PROGRAM main
VAR
	ButtonON_LED AT %IX100.0 : bool;
	ButtonOFF_LED AT %IX100.1 : bool;
	ButtonON_LEDBlink AT %IX100.2 : bool;
	ButtonOFF_LEDBlink AT %IX100.3 : bool;
	LED1 AT %QX100.0 : bool;
	LED2 AT %QX100.1 : bool;
	LED3 AT %QX100.2 : bool;
	Start_Blink : bool;
	TON0_Coil : bool;
	TON1_Coil : bool;
	TON0 : TON;
	TON1 : TON;
END_VAR

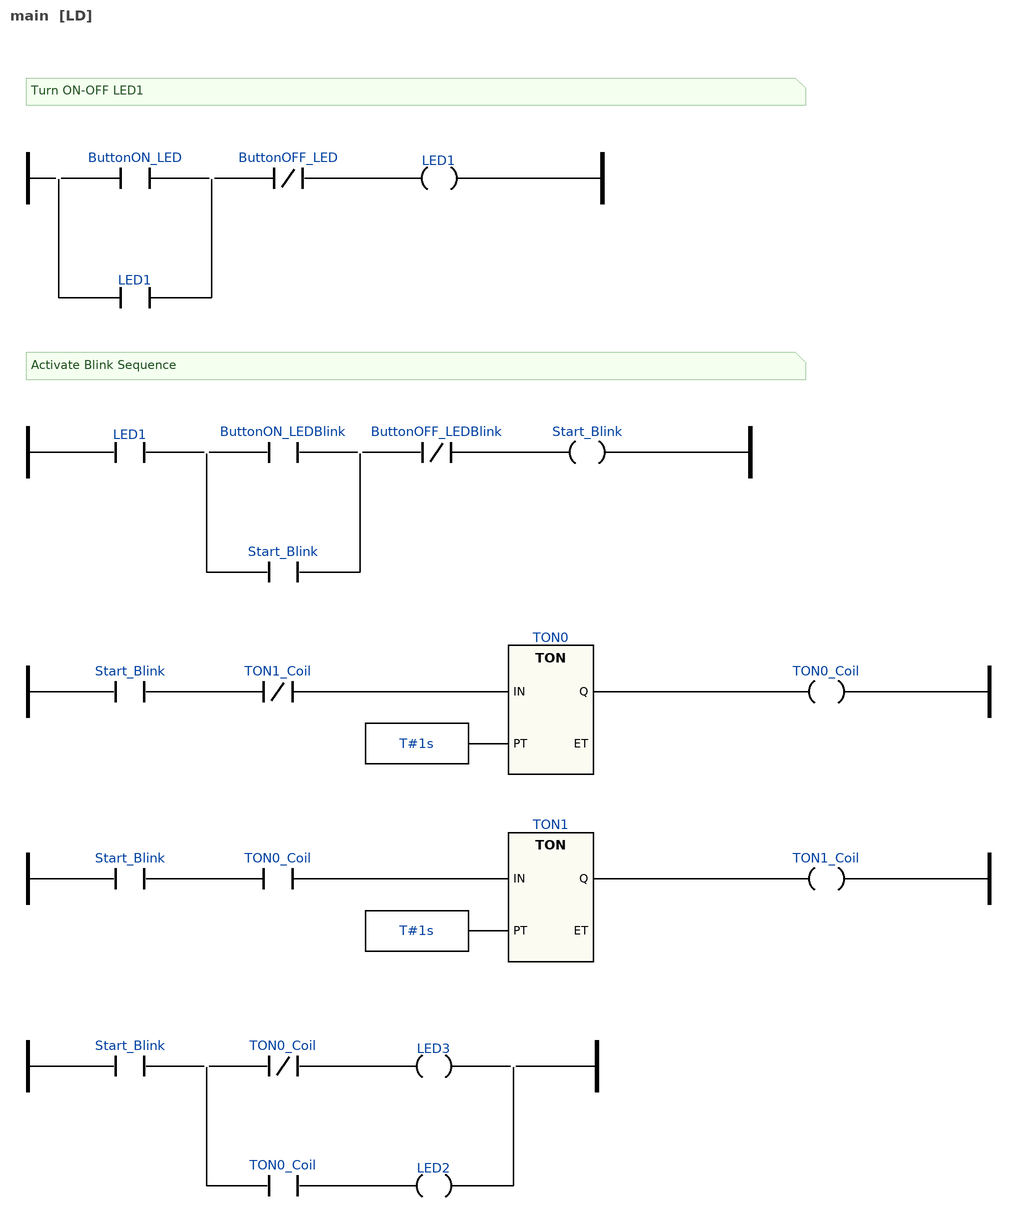
(* LD diagram, written out as Structured Text *)
(* Turn ON-OFF LED1 *)
LED1 := (ButtonON_LED OR LED1) AND NOT ButtonOFF_LED;
(* Activate Blink Sequence *)
Start_Blink := LED1 AND (ButtonON_LEDBlink OR Start_Blink) AND NOT ButtonOFF_LEDBlink;
TON0(IN := Start_Blink AND NOT TON1_Coil, PT := T#1s);
TON0_Coil := TON0.Q;
TON1(IN := Start_Blink AND TON0_Coil, PT := T#1s);
TON1_Coil := TON1.Q;
LED3 := Start_Blink AND NOT TON0_Coil;
LED2 := Start_Blink AND TON0_Coil;
END_PROGRAM
